PROGRAM P_ControlBlock
VAR
	fbDeadBandTester : FB_DeadbandTester;
	fbAutoClock : FB_AutoClock;
	fbMotionRef : FB_MotionRef;
	fbControl : FB_ControlSignal;
	fbInitialPos : FB_InitialPos;
END_VAR


fbControl(
	bFF := G_Enables.bEnableFF,
	bPID := G_Enables.bEnablePID,
	bU := G_Enables.bEnableU,
	bValve := TRUE,
	
	fDeadBandUp := G_Parameter.fDeadUp,
	fDeadBandDown := G_Parameter.fDeadDown
);


IF G_Mode.bAuto AND G_Mode.bRunning THEN

	fbInitialPos(
		bEnable := G_Inputs.bStartButton,
		fCurrentPos := G_OPC.fPistonPosition
	);
	
	fbAutoClock(
		fStart := G_Inputs.bStartButton,
		fRunning := G_Mode.bRunning,
		fCycle := G_Parameter.fCycleTime
	);
	
	fbMotionRef(
		fTime := fbAutoClock.fTime,
		fAmplitude := G_Parameter.fAmplitude,
		fInitialPos := fbInitialPos.fInitialPos,
		fFrequency := G_Parameter.fFrequency,
		fXDotRef => G_OPC.fXDotRef,
		fXRef => G_OPC.fXRef 
	);
	
	fbControl(
		fFF := G_OPC.fFF,
		fPID := G_OPC.fSignalPID,
		
		fU => G_OPC.fU
	);

ELSIF G_Mode.bManual AND G_Mode.bRunning THEN

	fbInitialPos(
		bEnable := G_Inputs.bStartButton,
		fCurrentPos := G_OPC.fPistonPosition
	);
	
	fbDeadBandTester(
		fInput := G_OPC.fJoystick,
		bEnable := TO_BOOL(G_Inputs.bManual),
		fConst := G_Parameter.fConst,
		fOutput => G_OPC.fU
	);


END_IF

END_PROGRAM

(* stored: Version 1.1.0.1, ProductVersion 3.1.4024.12
   POU P_ControlBlock: Id {34b73f17-fb3f-4014-8571-592d49402d29}, SpecialFunc None *)
